TEXTLIST TextList_Config_Chauffage
  0 = 'chauffage' | FR: 'CHAUFFAGE' | EN: 'HEATING'
  1 = 'PRM_Tp_Vent' | FR: 'Température max. pour ventilation enceinte' | EN: 'Max. temperature for chamber venting'
  2 = 'PRM_Max_Temp' | FR: 'Consigne température max.' | EN: 'Max. temperature setpoint'
  3 = 'CONF_Pmax' | FR: 'Puissance de chauffage max.' | EN: 'Max. heating setpoint'
  4 = 'P' | FR: 'Gain' | EN: 'Amplification factor'
  5 = 'Ti' | FR: "Temps d'action intégrale" | EN: 'Integral action time'
  6 = 'Td' | FR: "Temps d'action dérivée" | EN: 'Derivative action time'
  7 = 'Ta' | FR: "Temps d'amortissement" | EN: 'Damping time'
  8 = 'PRM_Border_Ratio' | FR: 'Coefficient de pondération chauffage bords' | EN: 'Border heating ratio'
  9 = 'Disable SD11' | FR: 'Désactivation thermocouple SD11' | EN: 'Disable SD11 thermocouple '
  10 = 'Disable SD12' | FR: 'Désactivation thermocouple SD12' | EN: 'Disable SD12 thermocouple '
  11 = 'Disable SD13' | FR: 'Désactivation thermocouple SD13' | EN: 'Disable SD13 thermocouple '
  12 = 'Disable SD14' | FR: 'Désactivation thermocouple SD14' | EN: 'Disable SD14 thermocouple '
  13 = 'Tc Ctrl' | FR: 'Thermocouples de régulation' | EN: 'Regulation thermocouples'
  14 = 'Tc Disp' | FR: 'Thermocouples de sécurité' | EN: 'Security thermocouples'
  15 = 'Tc conf' | FR: 'Configuration thermocouples' | EN: 'Thermocouples settings'
  16 = 'Temp min' | FR: 'Température min. avand défaut' | EN: 'Min. temperature before fault'
  17 = 'Temp max' | FR: 'Température max. avant défaut' | EN: 'Max temperature before fault'
  18 = 'Rechauf' | FR: 'Thermaliseur' | EN: 'Chiller'
   = ''
END_TEXTLIST

(* stored: Version 1.1.0.1, ProductVersion 3.1.4024.10
   TextList TextList_Config_Chauffage: Id {d160190e-db37-4f4d-aa83-3ba57e293aa6} *)
